{attribute 'linkalways'} 
{attribute 'no_explicit_call' := 'This FB is a CLASS and must be accessed using methods or properties'}
{attribute 'enable_dynamic_creation'}
FUNCTION_BLOCK StackDisposedEvent EXTENDS StackEvent IMPLEMENTS I_StackDisposedEvent

END_FUNCTION_BLOCK

(* stored: Version 1.1.0.1, ProductVersion 3.1.4024.12
   POU StackDisposedEvent: Id {ad473912-5b58-4634-97f4-438ae08e0a8e}, SpecialFunc None *)
